(* CODESYS project filling_station.ecp

Project tree, tasks and I/O mapping:
  GenericDummyMasterDevice : Generic Master, WAGO, order no. None, version 1.0.0.0
  PFC200_CS_2ETH_RS : 750-8202 PFC200 2ETH RS, WAGO, order no. 0750-8202, version 1.4.1.22
    application Application
      libraries: 
      task PLC_Task (cyclic, interval t#10ms, priority 14) calls PLC_PRG
      task VISU_TASK (cyclic, interval 100 ms, priority 15) calls VisuElems.Visu_Prg
      function CONVERT_PRESSURE_TO_LEVEL [ST]
      visualisation Visualization
      function READ_PRESSURE [ST]
      global variables GVL
      function XOR_MANUAL_AUTOMATIC_VALVE_CONTROL [ST]
      function STORE_LEVEL_HISTORY [ST]
      function SAMSON_VALVE_POSITION_CONTROLLER [ST]
      function READ_VALVE_POSITION [ST]
      function AVOID_SIMULT_VALVE_OPEN_AND_CLOSE [ST]
      program PLC_PRG [FBD]
      image pool ImagePool
      visualisation Visualization_detailed
    DeviceAdapter
    Kbus : Kbus, WAGO, version 1.3.0.0
        unmapped channels: K-BUS diagnostics
      _8_DO_Generic : 075x-8DO, WAGO, order no. 075x-8DO, version 0.0.0.11
          settings: K-BUS Module slot index = 1
          output vbOpenSamsonValve : BOOL  // _OUT._OUT
          output vbCloseSamsonValve : BOOL  // _OUT._OUT
          output vbOpenDrainValve : BOOL  // _OUT._OUT
          output vbSwitchOnPump : BOOL  // _OUT._OUT
          unmapped channels: _OUT
        DeviceAdapter
      _4_AI_0_10V_DC_s_e : 0750-0459, WAGO, order no. 0750-0459, version 0.0.0.11
          settings: K-BUS Module slot index = 2
          input  vwRawValvePosition : WORD  // _IW 1
          unmapped channels: _IW 2, _IW 3, _IW 4
        DeviceAdapter
      _2_AI_4_20mA_Diff_Measurement_Input : 0750-0492, WAGO, order no. 0750-0492, version 0.0.0.7
          settings: K-BUS Module slot index = 3
          input  vwRawPressure : WORD  // _IW 1
          unmapped channels: _IW 2
        DeviceAdapter
    MODBUS
      MODBUS : MODBUS, WAGO, order no. n/a, version 1.1.1.13
    Serial
      COM1 : COM1, WAGO, version 0.0.0.19
  e_DISPLAY_7300T_WP_10_1_1280x800_PIO1 : 0762-3003 e!DISPLAY 7300T - WP 10.1, WAGO, order no. 0762-3003, version 0.0.0.3
    DeviceAdapter
  libraries: WagoVisuIcons, 1.0.0.7 (WAGO)
  text list GlobalTextList
  5ce3da45-db07-42e7-a21c-a00fff4ed8f6|C:\Users\Alexander Wilms\Documents\Ausbildung\Hochschule Darmstadt\Master Electrical Engineering\1. Semester\Team Project\team-project\40_Implementation\hydraulics-schematic-simplified.png
  5ce3da45-db07-42e7-a21c-a00fff4ed8f6|C:\Users\Alexander Wilms\Documents\Ausbildung\Hochschule Darmstadt\Master Electrical Engineering\1. Semester\Team Project\team-project\30_Architecture\hydraulics-schematic-simplified.png
*)

// PFC200_CS_2ETH_RS/Application/GVL
VAR_GLOBAL
	vrWaterLevel:REAL;
	vrgrWaterLevel:ARRAY[1..16] OF REAL;
	vrStandardGravity:REAL:=9.81;
	viDensityWater:INT:=1000;
	vrValvePosition:REAL;
	vrValvePositionPercentage:REAL;
	vrValvePositionDesired:REAL;
	viPumpPowerPercentage:INT;
	vbManualValveControl:BOOL:=TRUE;
	vbAutomaticValveControl:BOOL:=FALSE;
	vbPreviousValveControl:STRING:='MANUAL';
	vbPreviousSamsonValveDirection:STRING:='STOP';
	vbStopSamsonValve:BOOL:=TRUE;
	vbOpenDrainValveBelowVessel:BOOL:=FALSE;
	vbOpenDrainValveAbovePump:BOOL:=FALSE;
	vbPowerOnPump:BOOL:=TRUE;
END_VAR

// PFC200_CS_2ETH_RS/Application/PLC_PRG
PROGRAM PLC_PRG
VAR
END_VAR
VAR // added by the converter: edge detectors and wires of the graphical bodies
    _w1 : REAL;
END_VAR

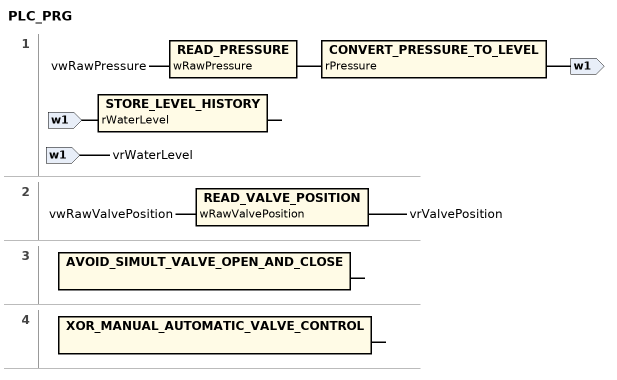
// NETWORK 1
_w1 := CONVERT_PRESSURE_TO_LEVEL(rPressure := READ_PRESSURE(wRawPressure := vwRawPressure));
STORE_LEVEL_HISTORY(rWaterLevel := _w1);
vrWaterLevel := _w1;

// NETWORK 2
vrValvePosition := READ_VALVE_POSITION(wRawValvePosition := vwRawValvePosition);

// NETWORK 3
AVOID_SIMULT_VALVE_OPEN_AND_CLOSE();

// NETWORK 4
XOR_MANUAL_AUTOMATIC_VALVE_CONTROL();

END_PROGRAM

// PFC200_CS_2ETH_RS/Application/CONVERT_PRESSURE_TO_LEVEL
FUNCTION CONVERT_PRESSURE_TO_LEVEL : REAL
VAR_INPUT
	rPressure:REAL;
END_VAR
VAR
END_VAR

CONVERT_PRESSURE_TO_LEVEL := rPressure/viDensityWater/vrStandardGravity;

END_FUNCTION

// PFC200_CS_2ETH_RS/Application/READ_PRESSURE
FUNCTION READ_PRESSURE : REAL
VAR_INPUT
	wRawPressure:WORD;
END_VAR
VAR
END_VAR

READ_PRESSURE := WORD_TO_REAL(wRawPressure)/65535*100000;

END_FUNCTION

// PFC200_CS_2ETH_RS/Application/STORE_LEVEL_HISTORY
FUNCTION STORE_LEVEL_HISTORY : BOOL
VAR_INPUT
	rWaterLevel:REAL;
END_VAR
VAR
	index: INT;
	rgrWaterLevelTmp:ARRAY[1..16] OF REAL;
	rgrWaterLevel: REAL;
END_VAR

rgrWaterLevelTmp := vrgrWaterLevel;

FOR index:=1 TO 15 DO
	vrgrWaterLevel[index]:= rgrWaterLevelTmp[index+1];
END_FOR

vrgrWaterLevel[16] := rWaterLevel;

END_FUNCTION

// PFC200_CS_2ETH_RS/Application/READ_VALVE_POSITION
FUNCTION READ_VALVE_POSITION : REAL
VAR_INPUT
	wRawValvePosition:WORD;
END_VAR
VAR
END_VAR

READ_VALVE_POSITION := WORD_TO_REAL(wRawValvePosition)/65535*1;
vrValvePositionPercentage := READ_VALVE_POSITION*100;

END_FUNCTION

// PFC200_CS_2ETH_RS/Application/AVOID_SIMULT_VALVE_OPEN_AND_CLOSE
FUNCTION AVOID_SIMULT_VALVE_OPEN_AND_CLOSE : BOOL
VAR_INPUT
END_VAR
VAR
END_VAR

IF vbOpenSamsonValve AND vbStopSamsonValve THEN
	IF vbPreviousSamsonValveDirection = 'OPEN' THEN
		vbOpenSamsonValve := FALSE;
		vbStopSamsonValve := TRUE;
		vbCloseSamsonValve := FALSE;
		vbPreviousSamsonValveDirection := 'STOP';
	ELSIF vbPreviousSamsonValveDirection = 'STOP' THEN
		vbOpenSamsonValve := TRUE;
		vbStopSamsonValve := FALSE;
		vbCloseSamsonValve := FALSE;
		vbPreviousSamsonValveDirection := 'OPEN';
	END_IF
ELSIF vbStopSamsonValve AND vbCloseSamsonValve THEN
	IF vbPreviousSamsonValveDirection = 'STOP' THEN
		vbOpenSamsonValve := FALSE;
		vbStopSamsonValve := FALSE;
		vbCloseSamsonValve := TRUE;
		vbPreviousSamsonValveDirection := 'CLOSE';
	ELSIF vbPreviousSamsonValveDirection = 'CLOSE' THEN
		vbOpenSamsonValve := FALSE;
		vbStopSamsonValve := TRUE;
		vbCloseSamsonValve := FALSE;
		vbPreviousSamsonValveDirection := 'STOP';
	END_IF
ELSIF vbOpenSamsonValve AND vbCloseSamsonValve THEN
	IF vbPreviousSamsonValveDirection = 'OPEN' THEN
		vbOpenSamsonValve := FALSE;
		vbStopSamsonValve := FALSE;
		vbCloseSamsonValve := TRUE;
		vbPreviousSamsonValveDirection := 'CLOSE';
	ELSIF vbPreviousSamsonValveDirection = 'CLOSE' THEN
		vbOpenSamsonValve := TRUE;
		vbStopSamsonValve := FALSE;
		vbCloseSamsonValve := FALSE;
		vbPreviousSamsonValveDirection := 'OPEN';
	END_IF
END_IF

AVOID_SIMULT_VALVE_OPEN_AND_CLOSE := TRUE;

END_FUNCTION

// PFC200_CS_2ETH_RS/Application/XOR_MANUAL_AUTOMATIC_VALVE_CONTROL
FUNCTION XOR_MANUAL_AUTOMATIC_VALVE_CONTROL : BOOL
VAR_INPUT
END_VAR
VAR
END_VAR

IF vbAutomaticValveControl AND vbManualValveControl THEN
	IF vbPreviousValveControl = 'MANUAL' THEN
			vbAutomaticValveControl := TRUE;
			vbManualValveControl := FALSE;
			vbPreviousValveControl := 'AUTOMATIC';
	ELSIF
			vbPreviousValveControl =  'AUTOMATIC' THEN
			vbAutomaticValveControl := FALSE;
			vbManualValveControl := TRUE;
			vbPreviousValveControl := 'MANUAL';
	END_IF
END_IF

XOR_MANUAL_AUTOMATIC_VALVE_CONTROL := TRUE;

END_FUNCTION

// PFC200_CS_2ETH_RS/Application/SAMSON_VALVE_POSITION_CONTROLLER
FUNCTION SAMSON_VALVE_POSITION_CONTROLLER : BOOL
VAR_INPUT
END_VAR
VAR
	delta:REAL:=0.1;
END_VAR

IF vbAutomaticValveControl = TRUE THEN
	IF vrValvePosition < vrValvePositionDesired/100 - delta THEN
		vbOpenSamsonValve := TRUE;
		vbSTOPSamsonValve := FALSE;
		vbCloseSamsonValve := FALSE;
		// this is just test code
		vrValvePosition := vrValvePosition + 0.01;
	ELSIF vrValvePosition > vrValvePositionDesired/100 + delta THEN
		vbOpenSamsonValve := FALSE;
		vbSTOPSamsonValve := FALSE;
		vbCloseSamsonValve := TRUE;
		// this is just test code
		vrValvePosition := vrValvePosition - 0.01;
	END_IF
END_IF

SAMSON_VALVE_POSITION_CONTROLLER := TRUE;

END_FUNCTION

// PFC200_CS_2ETH_RS/Application/Visualization
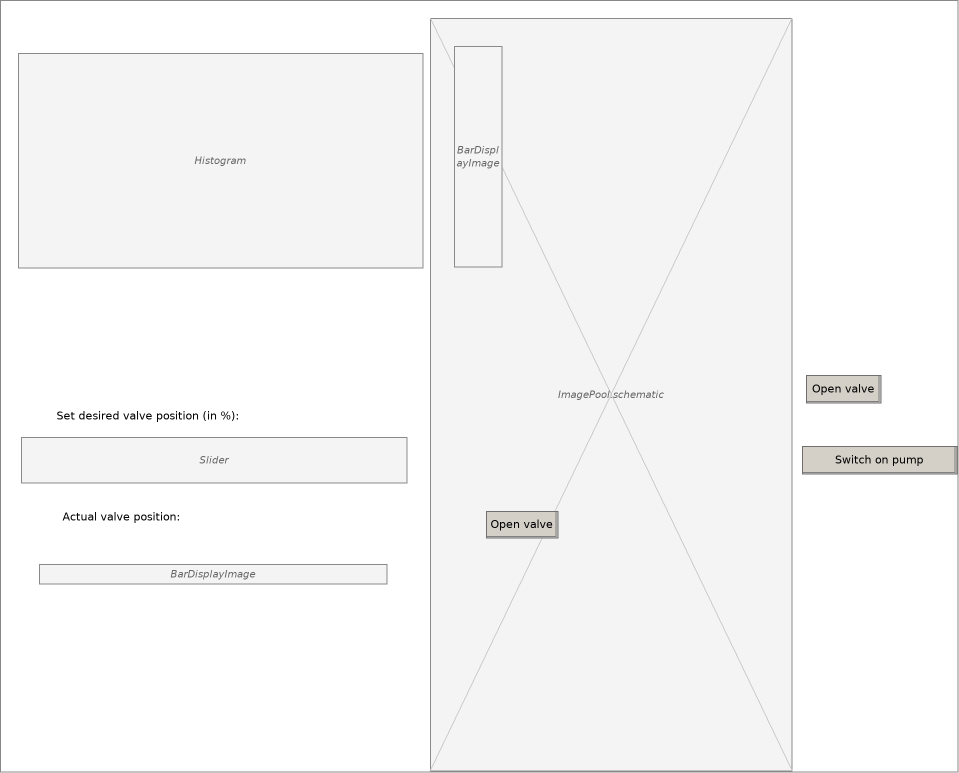
VISUALIZATION Visualization  // 959x773
    Image (430,18 362x753), image: ImagePool.schematic
    BarDisplayImage (454,46 48x221), value: vrWaterLevel, style: BarDisplayImage-Gray, scale format: %.1f, scale 0..1
        p518627256: m
    Histogram (18,53 405x215), scale format: %.1f, scale 0..1
        p1518820177: vrgrWaterLevel
        p102497268: vrgrWaterLevel
        p788070771: ARRAY [1..16] OF REAL
    Button (806,375 75x28), "Open valve"
        toggle vbOpenDrainValveAbovePump
    Button (802,446 155x28), "Switch on pump"
        toggle vbPowerOnPump
    Label (61,407 174x18), "Set desired valve position (in %):"
    Slider (21,437 386x46), variable: vrValvePositionDesired, scale 0..100
    Button (486,511 72x27), "Open valve"
        toggle vbOpenDrainValveBelowVessel
    BarDisplayImage (39,564 348x20), value: vrWaterLevel, style: BarDisplayImage-Gray, scale format: %i, scale 0..100
        p518627256: m
    Label (59,508 125x18), "Actual valve position:"
END_VISUALIZATION

// PFC200_CS_2ETH_RS/Application/Visualization_detailed
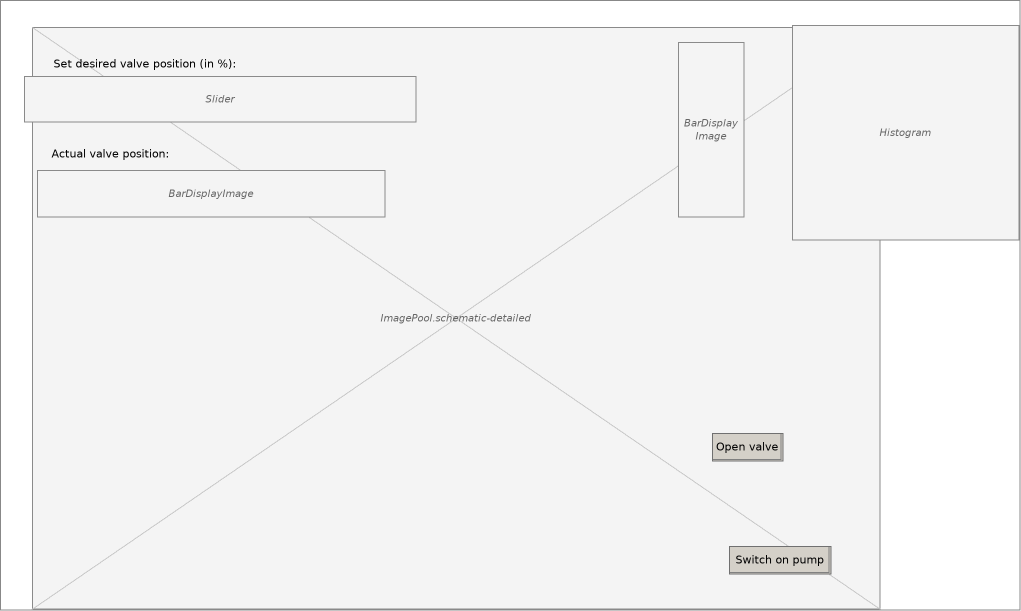
VISUALIZATION Visualization_detailed  // 1021x611
    Image (32,27 848x582), image: ImagePool.schematic-detailed
    BarDisplayImage (678,42 66x175), value: vrWaterLevel, style: BarDisplayImage-Gray, scale format: %.1f, scale 0..1
        p518627256: m
    Histogram (792,25 227x215), scale format: %.1f, scale 0..1
        p1518820177: vrgrWaterLevel
        p102497268: vrgrWaterLevel
        p788070771: ARRAY [1..16] OF REAL
    Button (712,433 71x28), "Open valve"
        toggle vbOpenDrainValveAbovePump
    Button (729,546 102x28), "Switch on pump"
        toggle vbPowerOnPump
    Label (58,55 174x18), "Set desired valve position (in %):"
    Slider (24,76 392x46), variable: vrValvePositionDesired, scale 0..100
    BarDisplayImage (37,170 348x47), value: vrWaterLevel, style: BarDisplayImage-Gray, scale format: %i, scale 0..100
        p518627256: m
    Label (48,145 125x18), "Actual valve position:"
END_VISUALIZATION
